Staubli VAL3: onF1Event.pgx

program onF1Event()
  local num l
begin
  // look if the bButton is enable
  if bButton[0]
    //
    // go to previous POINT
    //
    if !cycleStatus:bCycle or !cycleStatus:bSimulation
      call goTo(nPoint-1)
    endIf
  endIf
end
